// TwinCAT 3 PLC project PLC1
// ProgramVersion: 3.1.4023.0
// libraries:
//   Tc2_Standard, * (Beckhoff Automation GmbH)
//   Tc2_System, * (Beckhoff Automation GmbH)
//   Tc3_Module, * (Beckhoff Automation GmbH)
// project tree:
//   GVLs/ GVL.TcGVL
//   / PlcTask.TcTTO
//   POUs/ MAIN.TcPOU
// real-time tasks:
//   TASK PlcTask: cycle T#10ms, priority 20, ADS port 350
// motion (NC):
//   TASK NC-Task 1 SAF: cycle T#2ms, priority 4, ADS port 501
//   TASK NC-Task 1 SVB: cycle T#10ms, priority 8, ADS port 511
//   AXIS Axis 1 (id 1)
//     General: UnitName=Degree
//     OtherSettings: AllowMotionCmdToSlave=true
//     encoder EncType=19
//       EncPara: ScaleFactorNumerator=360, ScaleFactorDenominator=8000, MaxCount=#xffffffff
//     drive DrvType=16
//       DrvPara: MaxCount=#xffffffff
//         Analog: TorqueSetpointScale=10, ScaleFactorActTorque=0.1
//         TimeComp: TaskDelayCycles=1
//     controller CtrType=1
//       CtrPara: PriorControlFactor=1
//         Observer: BandWidth=20
// I/O:
//   DEVICE Device 1 (EtherCAT), AmsNetId 5.72.219.114.2.1
//     Term 1 (EK1200) [EK1200-5000 EtherCAT Power supply (2A E-Bus)]
//       Term 2 (EL6751) [EL6751 CANopen Master]
//       Term 3 (EL9011) [EL9011 End Terminal]
//   DEVICE Device 4 (EL6751), AmsNetId 5.72.219.114.5.1
//     Box 5 JAT (CANopen Node)
// variable links:
//   PLC1/PLC1 Instance <-> Device 4 (EL6751)/Box 5 JAT (CANopen Node)
//     PlcTask Inputs/GVL.ModesOfOperationDisplay <-> TxPDO 1/Inputs/ModesOfOperationDisplay
//     PlcTask Inputs/GVL.Statuswort <-> TxPDO 1/Inputs/Statuswort
//     PlcTask Inputs/GVL.digital_inputs_jat <-> TxPDO 1/Inputs/digital_inputs_jat
//     PlcTask Inputs/GVL.pos_actual_value <-> TxPDO 1/Inputs/pos_actual_value
//     PlcTask Inputs/GVL.velocity_actual_value <-> TxPDO 2/Inputs/velocity_actual_value
//     PlcTask Inputs/GVL.velocity_sensor_actual_value <-> TxPDO 2/Inputs/velocity_sensor_actual_value
//     PlcTask Outputs/GVL.Kontrollwort <-> RxPDO 1/Outputs/Kontrollwort
//     PlcTask Outputs/GVL.ModesOfOperation <-> RxPDO 1/Outputs/ModesOfOperation
//     PlcTask Outputs/GVL.pos_demand_value <-> RxPDO 1/Outputs/pos_demand_value
//     PlcTask Outputs/GVL.profile_acceleration <-> RxPDO 2/Outputs/profile_acceleration
//     PlcTask Outputs/GVL.profile_deceleration <-> RxPDO 3/Outputs/profile_deceleration
//     PlcTask Outputs/GVL.profile_velocity <-> RxPDO 2/Outputs/profile_velocity
//     PlcTask Outputs/GVL.s_digital_inputs_jat <-> RxPDO 1/Outputs/s_digital_outputs_jat

CONFIGURATION PLC1
    RESOURCE PLC ON TwinCAT3
        TASK PlcTask(INTERVAL := T#10ms, PRIORITY := 20);
        PROGRAM MAIN WITH PlcTask : MAIN;
    END_RESOURCE
END_CONFIGURATION

// ---- GVLs/GVL.TcGVL
VAR_GLOBAL PERSISTENT
	// Test IO
	Statuswort								AT %I* : WORD;
	pos_actual_value 						AT %I* : DINT;
	ModesOfOperationDisplay					AT %I* : BYTE;
	digital_inputs_jat						AT %I* : BYTE;
	velocity_actual_value					AT %I* : DINT;
	velocity_sensor_actual_value			AT %I* : DINT;
	                                		
	Kontrollwort    						AT %Q* : WORD;
	pos_demand_value						AT %Q* : DINT;
	ModesOfOperation						AT %Q* : BYTE;
	s_digital_inputs_jat					AT %Q* : BYTE;
	profile_velocity						AT %Q* : DINT;
	profile_acceleration					AT %Q* : DINT;
	profile_deceleration					AT %Q* : DINT;
END_VAR

// ---- POUs/MAIN.TcPOU
PROGRAM MAIN
VAR
END_VAR

END_PROGRAM
